FUNCTION_BLOCK Sensor_Bool_CAT (* Composite Function Block Type *)
  (* Standard: 61499-2 *)
  (* Version 0.0, 2/2/2026, Schneider Electric, template *)
  PACKAGE Main;
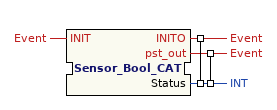
  EVENT_INPUT
    INIT; (* Initialization Request *)
  END_EVENT
  EVENT_OUTPUT
    INITO WITH Status; (* Initialization Confirm *)
    pst_out WITH Status; (* Execution Confirmation *)
  END_EVENT
  VAR_OUTPUT
    Status : INT; (* Output event qualifier *)
  END_VAR
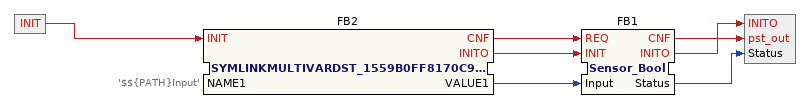
  FBS
    FB1 : Sensor_Bool;
    FB2 : SYMLINKMULTIVARDST_1559B0FF8170C9BA0(NAME1 := '$${PATH}Input'); {SET_ATTRIBUTE(Configuration.GenericFBType.InterfaceParams, Runtime.System#I:=1;VALUE${I$}:BOOL)}
  END_FBS
  EVENT_CONNECTIONS
    FB2.CNF TO FB1.REQ;
    FB2.INITO TO FB1.INIT;
    INIT TO FB2.INIT;
    FB1.CNF TO pst_out;
    FB1.INITO TO INITO;
  END_CONNECTIONS
  DATA_CONNECTIONS
    FB2.VALUE1 TO FB1.Input;
    FB1.Status TO Status;
  END_CONNECTIONS
END_FUNCTION_BLOCK
